Universal Robots PolyScope program: rtde_control_loop_2.urp

Program rtde_control_loop_2 (installation=default directory=/programs/usbdisk/reconhecimento_mao createdIn=3.2.19275.0 lastSavedIn=5.9.4.1031232 robotSerialNumber=20185500417)
Calibrated DH parameters: a=[0.000198, -0.213715, -0.379508, 0.000129, 0.000086, 0]; d=[0.162607, 159.179056, -212.880985, 53.835388, 0.099715, 0.099672]; alpha=[1.570039, -0.002309, 0.001844, 1.570423, -1.570488, 0]; deltaTheta=[0, -1.044161, 7.072154, 0.255189, 0, 0]
BeforeStart
  setp := Joint_6_name
  Script: rtde_set_watchdog("input_int_register_0", 1, "PAUSE")
  MoveJ speed 60 deg/s, acceleration 80 deg/s^2 (useActiveTCP=true) feature=Base
    Waypoint Waypoint_1: TCP in base x=452.093 y=-173.437 z=680.935 mm, rx=1.2913 ry=1.1488 rz=1.0964 rad; joints [0.055, -51.715, -113.816, -16.795, 82.796, 0.022] deg; TCP offset x=0 y=0 z=234.35 mm, rx=0 ry=0 rz=-3.1416 rad
    tmp := p[0.21967,-0.1476,0.6,-1.18093,1.32761,-1.282]
    Script: sync()
Robot Program (runOnlyOnce=false)
  Loop Forever
    SuppressedNode
      var_2 := read_input_integer_register(8)
    SuppressedNode
      Switch expression=var_2
        Case (caseValue=10)
          MoveJ speed 60 deg/s, acceleration 80 deg/s^2 (useActiveTCP=true) feature=Base
            Waypoint Waypoint_1: TCP in base x=452.093 y=-173.437 z=680.935 mm, rx=1.2913 ry=1.1488 rz=1.0964 rad; joints [0.055, -51.715, -113.816, -16.795, 82.796, 0.022] deg
        Case (caseValue=20)
          MoveL speed 600 mm/s, acceleration 1200 mm/s^2 (useActiveTCP=true) feature=Base
            Waypoint Waypoint_2: TCP in base x=452.121 y=-173.35 z=841.551 mm, rx=1.2912 ry=1.1489 rz=1.0965 rad; joints [0.193, -60.77, -84.869, -36.684, 82.714, 0.002] deg; TCP offset x=0 y=0 z=234.35 mm, rx=0 ry=0 rz=-3.1416 rad
    SuppressedNode
      Switch expression=var_1
        Case (caseValue=11)
          Set DigitalOutput pin=digital_out[4]; digitalValue=1
        Case (caseValue=21)
          Set DigitalOutput pin=digital_out[4]; digitalValue=0
    MoveL speed 500 mm/s, acceleration 500 mm/s^2 (useActiveTCP=false) tcp=TCP_mao; feature=Base
      SuppressedNode
        Waypoint Waypoint_3: TCP in base x=386.788 y=-144.63 z=727.346 mm, rx=-1.0613 ry=1.2174 rz=-1.3432 rad; joints [0.095, -77.606, -96.647, 0.604, 82.796, 0.023] deg
      Waypoint Waypoint (Variable): variable=tmp
      Wait Sleep waitTime=0.1
    Script: sync()
  SuppressedNode
    Script: write_output_integer_register(0, 0)
  SuppressedNode
    Script: sync()
  SuppressedNode
    Script: write_output_integer_register(0, 1)
Thread Thread_1 (runOnlyOnce=false)
  setp := Joint_6_name
  Loop Forever
    var_1 := read_input_integer_register(7)
    tmp := p[0,0,0,0,0,0]
    Script: tmp[0] = read_input_float_register(0)
    Script: tmp[1] = read_input_float_register(1)
    Script: tmp[2] = read_input_float_register(2)
    Script: tmp[3] = read_input_float_register(3)
    Script: tmp[4] = read_input_float_register(4)
    Script: tmp[5] = read_input_float_register(5)
    var_4 := get_actual_tcp_pose()
    Switch expression=var_1
      Case (caseValue=11)
        URCap RG6 (RG - On Robot, OnRobot A/S) dataModel(depthCompensate=false, payload=0.0, force=25, width=10, name=RG6(10))
      Case (caseValue=21)
        URCap RG6 (RG - On Robot, OnRobot A/S) dataModel(depthCompensate=false, payload=0.0, force=25, width=70, name=RG6(70))
    SuppressedNode
      If tmp != p[0,0,0,0,0,0]
        setp := tmp
    Script: sync()
